// TIA Portal V19 export
TYPE "LEXCHANGETRAY_typeAxisSimpleControlCommandConfiguration2"
// stored: Access Published
   STRUCT
      power { S7_SetPoint := 'True'} : "LBC_typeAxisSimpleControlPower";
      reset { S7_SetPoint := 'True'} : "LBC_typeAxisSimpleControlReset";
      home { S7_SetPoint := 'True'} : "LBC_typeAxisSimpleControlHome";
      halt { S7_SetPoint := 'True'} : "LBC_typeAxisSimpleControlHalt";
      posAbsolute { S7_SetPoint := 'True'} : "LBC_typeAxisSimpleControlMoveAbsolute";
      posRelative { S7_SetPoint := 'True'} : "LBC_typeAxisSimpleControlMoveRelative";
      moveVelocity { S7_SetPoint := 'True'} : "LBC_typeAxisSimpleControlMoveVelocity";
      jog { S7_SetPoint := 'True'} : "LBC_typeAxisSimpleControlMoveJog";
      stop { S7_SetPoint := 'True'} : "LBC_typeAxisSimpleControlStop";
      readValues { S7_SetPoint := 'True'} : "LBC_typeAxisSimpleControlReadValues";
      torqueLimit { S7_SetPoint := 'True'} : "LEXCHANGETRAY_typeAxisSimpleControlTorqueLimit";
   END_STRUCT;
END_TYPE
